// Mitsubishi GX Works2 project: AutoStatisticWorkTime   PLC: FX3U/FX3UC

PROGRAM MAIN
VAR
  XO46 : BOOL;
END_VAR
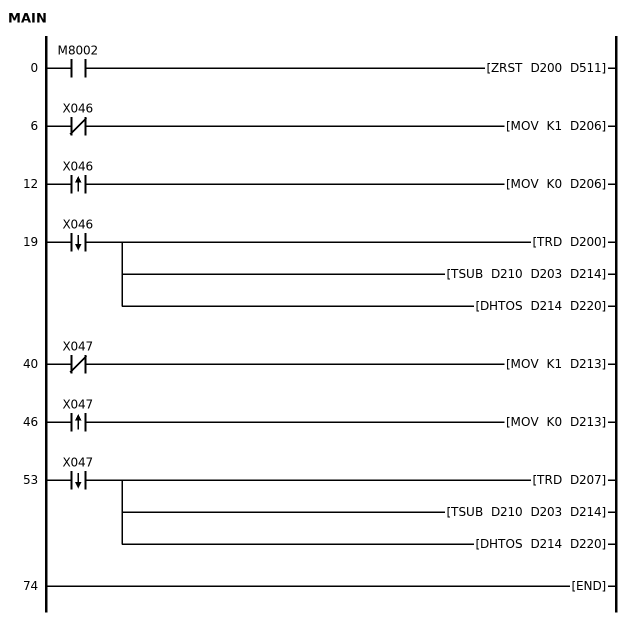
0     LD      M8002
      ZRST    D200 D511
6     LDI     X046
      MOV     K1 D206
12    LDP     X046
      MOV     K0 D206
19    LDF     X046
      TRD     D200
      TSUB    D210 D203 D214
      DHTOS   D214 D220
40    LDI     X047
      MOV     K1 D213
46    LDP     X047
      MOV     K0 D213
53    LDF     X047
      TRD     D207
      TSUB    D210 D203 D214
      DHTOS   D214 D220
74    END
END_PROGRAM
